Staubli VAL3: check_out_set.pgx

program check_out_set(dio x_dDio_target, bool x_bBool_onoff)
begin
  if ioStatus(x_dDio_target) >= 0
    //once io is working
    x_dDio_target = x_bBool_onoff
  endIf
end
